// Mitsubishi GX Works2 project: 01.CumBT   PLC: FX3U/FX3UC

// global labels: Global1
VAR_GLOBAL
  Clock_Sys : INT;
  IsServer : BOOL;
  D_ReadCode : TIMER;
  D_Output : TIMER;
  OK_NG : INT;
END_VAR

FUNCTION_BLOCK Check_QR_Code
VAR_INPUT
  Req : BOOL;
END_VAR
VAR_OUTPUT
  Done : BOOL;
  Busy : BOOL;
  Error : INT;
  Trigger : BOOL;
  S_Code : INT;
END_VAR
VAR_IN_OUT
  CheckDone : BOOL;
  CfOK : INT;
END_VAR
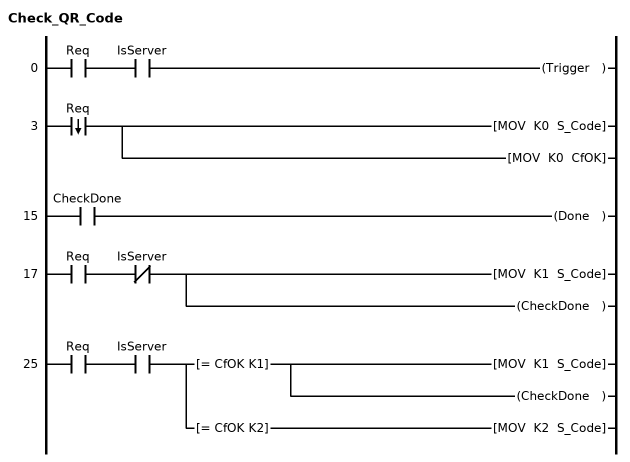
0     LD      Req
      AND     IsServer
      OUT     Trigger
3     LDF     Req
      MOV     K0 S_Code
      MOV     K0 CfOK
15    LD      CheckDone
      OUT     Done
17    LD      Req
      ANI     IsServer
      MOV     K1 S_Code
      OUT     CheckDone
25    LD      Req
      AND     IsServer
      MPS
      AND=    CfOK K1
      MOV     K1 S_Code
      OUT     CheckDone
      MPP
      AND=    CfOK K2
      MOV     K2 S_Code
END_FUNCTION_BLOCK

FUNCTION_BLOCK Control_Machine
VAR_INPUT
  AM : BOOL;
END_VAR
VAR_OUTPUT
  Red : BOOL;
  Yellow : BOOL;
  Green : BOOL;
  Buzz : BOOL;
  FlagRun : BOOL;
END_VAR
END_FUNCTION_BLOCK

FUNCTION_BLOCK Conveyer
VAR_INPUT
  AM : BOOL;
  EMG : BOOL;
END_VAR
VAR_OUTPUT
  Run_FWD : BOOL;
  Stopper_1_Up : BOOL;
  Stopper_1_Down : BOOL;
  Stopper_2_Up : BOOL;
  Stopper_2_Down : BOOL;
  Stopper_3_Up : BOOL;
  Stopper_3_Down : BOOL;
  Stopper_4_Up : BOOL;
  Stopper_4_Down : BOOL;
  XL_Up_Jig : BOOL;
  XL_Down_Jig : BOOL;
  Error_Code : INT;
END_VAR
VAR
  M_U_S1 : BOOL;
  M_D_S1 : BOOL;
  M_S_Stp1 : INT;
  M_U_S2 : BOOL;
  M_D_S2 : BOOL;
  M_S_Stp2 : INT;
  M_U_S3 : BOOL;
  M_D_S3 : BOOL;
  M_S_Stp3 : INT;
  M_U_S4 : BOOL;
  M_D_S4 : BOOL;
  M_S_Stp4 : INT;
  M_U_Jig : BOOL;
  M_D_Jig : BOOL;
  M_S_Cyl_J : INT;
  M_FWD : BOOL;
END_VAR
VAR_INPUT
  I_M_U_S1 : BOOL;
  I_M_D_S1 : BOOL;
  I_M_U_S2 : BOOL;
  I_M_D_S2 : BOOL;
  I_M_U_S3 : BOOL;
  I_M_D_S3 : BOOL;
  I_M_U_S4 : BOOL;
  I_M_D_S4 : BOOL;
  I_M_U_Jig : BOOL;
  I_M_D_Jig : BOOL;
  I_M_FWD : BOOL;
  I_M_Stop : BOOL;
END_VAR
VAR
  A_U_S1 : BOOL;
  A_D_S1 : BOOL;
  A_U_S2 : BOOL;
  A_D_S2 : BOOL;
  A_U_S3 : BOOL;
  A_D_S3 : BOOL;
  A_U_S4 : BOOL;
  A_D_S4 : BOOL;
  A_U_J : BOOL;
  A_D_J : BOOL;
END_VAR
VAR_INPUT
  A_S_Stp1 : INT;
  A_S_Stp2 : INT;
  A_S_Stp3 : INT;
  A_S_Stp4 : INT;
  A_S_Cyl_J : INT;
  A_FWD : BOOL;
END_VAR
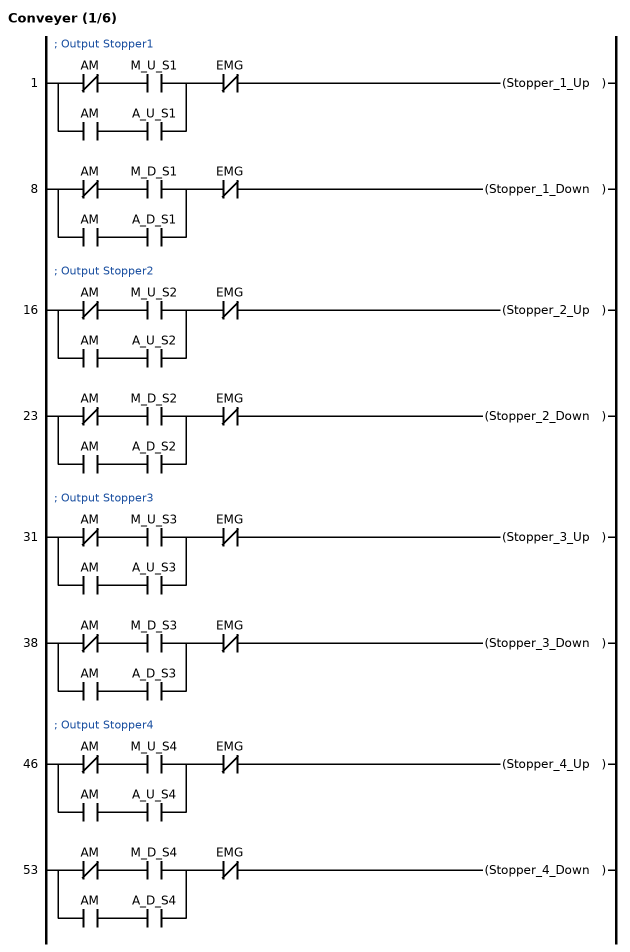
; Output Stopper1
1     LDI     AM
      AND     M_U_S1
      LD      AM
      AND     A_U_S1
      ORB
      ANI     EMG
      OUT     Stopper_1_Up
8     LDI     AM
      AND     M_D_S1
      LD      AM
      AND     A_D_S1
      ORB
      ANI     EMG
      OUT     Stopper_1_Down
; Output Stopper2
16    LDI     AM
      AND     M_U_S2
      LD      AM
      AND     A_U_S2
      ORB
      ANI     EMG
      OUT     Stopper_2_Up
23    LDI     AM
      AND     M_D_S2
      LD      AM
      AND     A_D_S2
      ORB
      ANI     EMG
      OUT     Stopper_2_Down
; Output Stopper3
31    LDI     AM
      AND     M_U_S3
      LD      AM
      AND     A_U_S3
      ORB
      ANI     EMG
      OUT     Stopper_3_Up
38    LDI     AM
      AND     M_D_S3
      LD      AM
      AND     A_D_S3
      ORB
      ANI     EMG
      OUT     Stopper_3_Down
; Output Stopper4
46    LDI     AM
      AND     M_U_S4
      LD      AM
      AND     A_U_S4
      ORB
      ANI     EMG
      OUT     Stopper_4_Up
53    LDI     AM
      AND     M_D_S4
      LD      AM
      AND     A_D_S4
      ORB
      ANI     EMG
      OUT     Stopper_4_Down
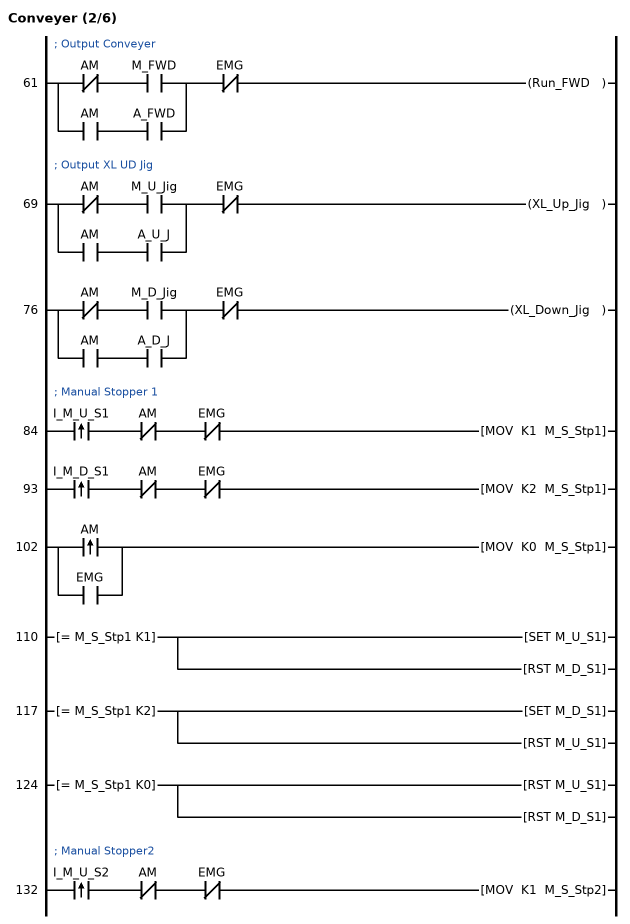
; Output Conveyer
61    LDI     AM
      AND     M_FWD
      LD      AM
      AND     A_FWD
      ORB
      ANI     EMG
      OUT     Run_FWD
; Output XL UD Jig
69    LDI     AM
      AND     M_U_Jig
      LD      AM
      AND     A_U_J
      ORB
      ANI     EMG
      OUT     XL_Up_Jig
76    LDI     AM
      AND     M_D_Jig
      LD      AM
      AND     A_D_J
      ORB
      ANI     EMG
      OUT     XL_Down_Jig
; Manual Stopper 1
84    LDP     I_M_U_S1
      ANI     AM
      ANI     EMG
      MOV     K1 M_S_Stp1
93    LDP     I_M_D_S1
      ANI     AM
      ANI     EMG
      MOV     K2 M_S_Stp1
102   LDP     AM
      OR      EMG
      MOV     K0 M_S_Stp1
110   LD=     M_S_Stp1 K1
      SET     M_U_S1
      RST     M_D_S1
117   LD=     M_S_Stp1 K2
      SET     M_D_S1
      RST     M_U_S1
124   LD=     M_S_Stp1 K0
      RST     M_U_S1
      RST     M_D_S1
; Manual Stopper2
132   LDP     I_M_U_S2
      ANI     AM
      ANI     EMG
      MOV     K1 M_S_Stp2
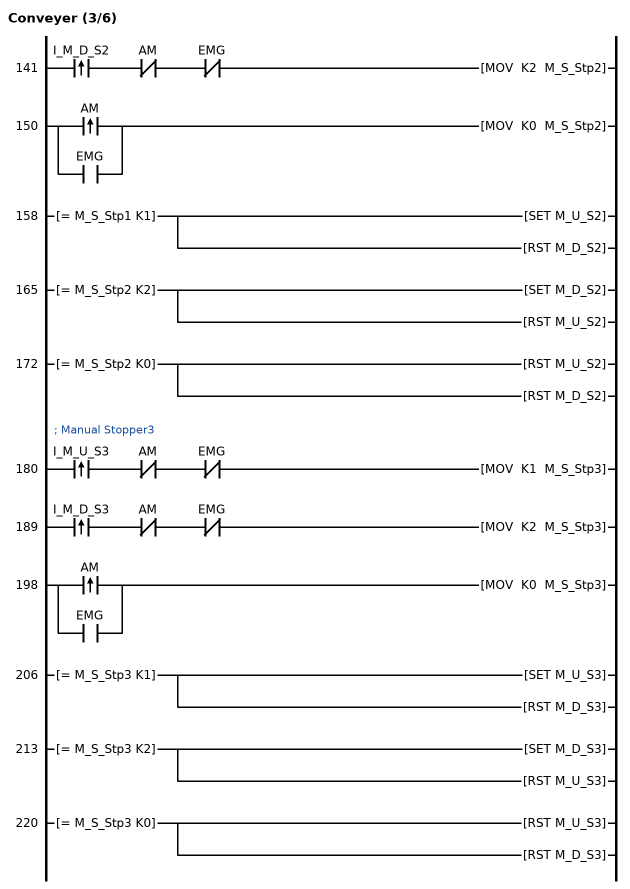
141   LDP     I_M_D_S2
      ANI     AM
      ANI     EMG
      MOV     K2 M_S_Stp2
150   LDP     AM
      OR      EMG
      MOV     K0 M_S_Stp2
158   LD=     M_S_Stp1 K1
      SET     M_U_S2
      RST     M_D_S2
165   LD=     M_S_Stp2 K2
      SET     M_D_S2
      RST     M_U_S2
172   LD=     M_S_Stp2 K0
      RST     M_U_S2
      RST     M_D_S2
; Manual Stopper3
180   LDP     I_M_U_S3
      ANI     AM
      ANI     EMG
      MOV     K1 M_S_Stp3
189   LDP     I_M_D_S3
      ANI     AM
      ANI     EMG
      MOV     K2 M_S_Stp3
198   LDP     AM
      OR      EMG
      MOV     K0 M_S_Stp3
206   LD=     M_S_Stp3 K1
      SET     M_U_S3
      RST     M_D_S3
213   LD=     M_S_Stp3 K2
      SET     M_D_S3
      RST     M_U_S3
220   LD=     M_S_Stp3 K0
      RST     M_U_S3
      RST     M_D_S3
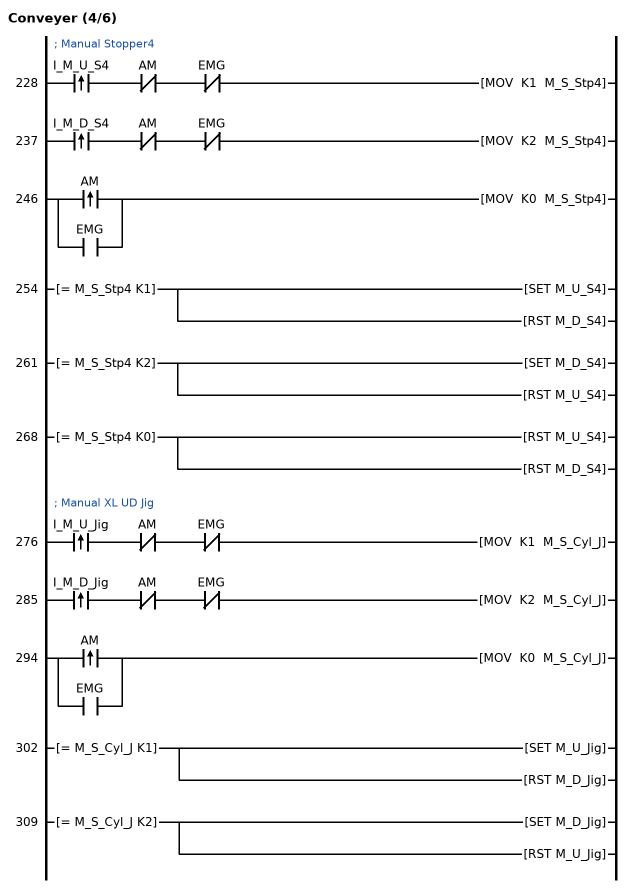
; Manual Stopper4
228   LDP     I_M_U_S4
      ANI     AM
      ANI     EMG
      MOV     K1 M_S_Stp4
237   LDP     I_M_D_S4
      ANI     AM
      ANI     EMG
      MOV     K2 M_S_Stp4
246   LDP     AM
      OR      EMG
      MOV     K0 M_S_Stp4
254   LD=     M_S_Stp4 K1
      SET     M_U_S4
      RST     M_D_S4
261   LD=     M_S_Stp4 K2
      SET     M_D_S4
      RST     M_U_S4
268   LD=     M_S_Stp4 K0
      RST     M_U_S4
      RST     M_D_S4
; Manual XL UD Jig
276   LDP     I_M_U_Jig
      ANI     AM
      ANI     EMG
      MOV     K1 M_S_Cyl_J
285   LDP     I_M_D_Jig
      ANI     AM
      ANI     EMG
      MOV     K2 M_S_Cyl_J
294   LDP     AM
      OR      EMG
      MOV     K0 M_S_Cyl_J
302   LD=     M_S_Cyl_J K1
      SET     M_U_Jig
      RST     M_D_Jig
309   LD=     M_S_Cyl_J K2
      SET     M_D_Jig
      RST     M_U_Jig
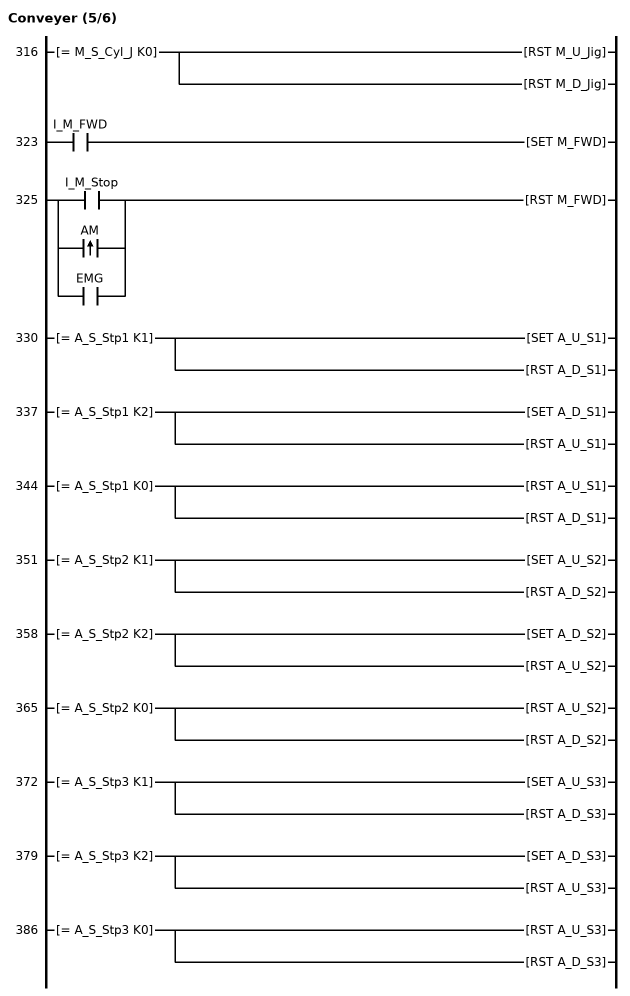
316   LD=     M_S_Cyl_J K0
      RST     M_U_Jig
      RST     M_D_Jig
323   LD      I_M_FWD
      SET     M_FWD
325   LD      I_M_Stop
      ORP     AM
      OR      EMG
      RST     M_FWD
330   LD=     A_S_Stp1 K1
      SET     A_U_S1
      RST     A_D_S1
337   LD=     A_S_Stp1 K2
      SET     A_D_S1
      RST     A_U_S1
344   LD=     A_S_Stp1 K0
      RST     A_U_S1
      RST     A_D_S1
351   LD=     A_S_Stp2 K1
      SET     A_U_S2
      RST     A_D_S2
358   LD=     A_S_Stp2 K2
      SET     A_D_S2
      RST     A_U_S2
365   LD=     A_S_Stp2 K0
      RST     A_U_S2
      RST     A_D_S2
372   LD=     A_S_Stp3 K1
      SET     A_U_S3
      RST     A_D_S3
379   LD=     A_S_Stp3 K2
      SET     A_D_S3
      RST     A_U_S3
386   LD=     A_S_Stp3 K0
      RST     A_U_S3
      RST     A_D_S3
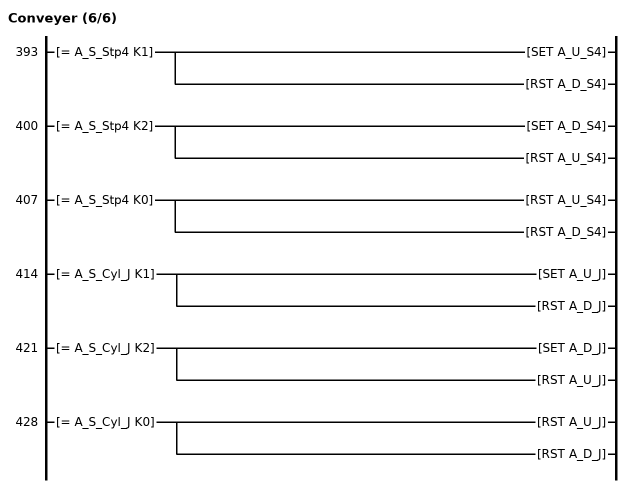
393   LD=     A_S_Stp4 K1
      SET     A_U_S4
      RST     A_D_S4
400   LD=     A_S_Stp4 K2
      SET     A_D_S4
      RST     A_U_S4
407   LD=     A_S_Stp4 K0
      RST     A_U_S4
      RST     A_D_S4
414   LD=     A_S_Cyl_J K1
      SET     A_U_J
      RST     A_D_J
421   LD=     A_S_Cyl_J K2
      SET     A_D_J
      RST     A_U_J
428   LD=     A_S_Cyl_J K0
      RST     A_U_J
      RST     A_D_J
END_FUNCTION_BLOCK

PROGRAM Data
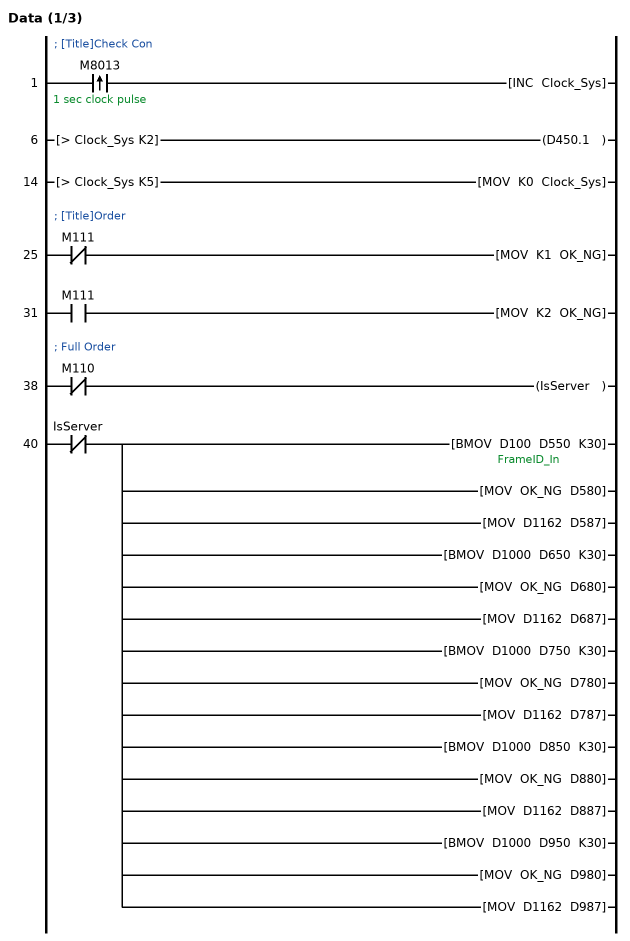
; [Title]Check Con
1     LDP     M8013  ; 1 sec clock pulse
      INC     Clock_Sys
6     LD>     Clock_Sys K2
      OUT     D450.1
14    LD>     Clock_Sys K5
      MOV     K0 Clock_Sys
; [Title]Order
25    LDI     M111
      MOV     K1 OK_NG
31    LD      M111
      MOV     K2 OK_NG
; Full Order
38    LDI     M110
      OUT     IsServer
40    LDI     IsServer
      BMOV    D100 D550 K30  ; FrameID_In
      MOV     OK_NG D580
      MOV     D1162 D587
      BMOV    D1000 D650 K30
      MOV     OK_NG D680
      MOV     D1162 D687
      BMOV    D1000 D750 K30
      MOV     OK_NG D780
      MOV     D1162 D787
      BMOV    D1000 D850 K30
      MOV     OK_NG D880
      MOV     D1162 D887
      BMOV    D1000 D950 K30
      MOV     OK_NG D980
      MOV     D1162 D987
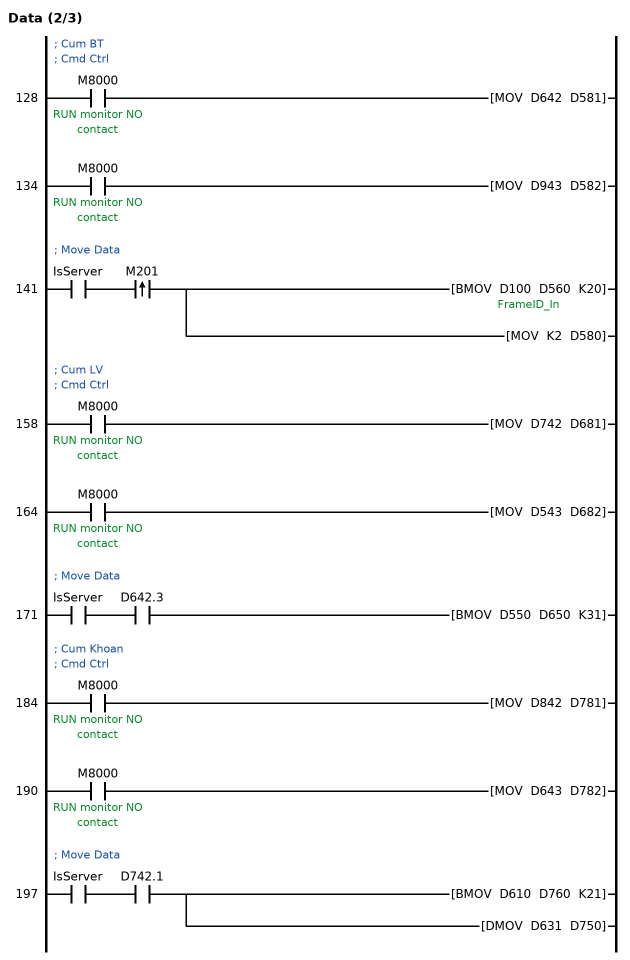
; Cum BT
; Cmd Ctrl
128   LD      M8000  ; RUN monitor NO contact
      MOV     D642 D581
134   LD      M8000  ; RUN monitor NO contact
      MOV     D943 D582
; Move Data
141   LD      IsServer
      ANDP    M201
      BMOV    D100 D560 K20
      MOV     K2 D580
; Cum LV
; Cmd Ctrl
158   LD      M8000  ; RUN monitor NO contact
      MOV     D742 D681
164   LD      M8000  ; RUN monitor NO contact
      MOV     D543 D682
; Move Data
171   LD      IsServer
      AND     D642.3
      BMOV    D550 D650 K31
; Cum Khoan
; Cmd Ctrl
184   LD      M8000  ; RUN monitor NO contact
      MOV     D842 D781
190   LD      M8000  ; RUN monitor NO contact
      MOV     D643 D782
; Move Data
197   LD      IsServer
      AND     D742.1
      BMOV    D610 D760 K21
      DMOV    D631 D750
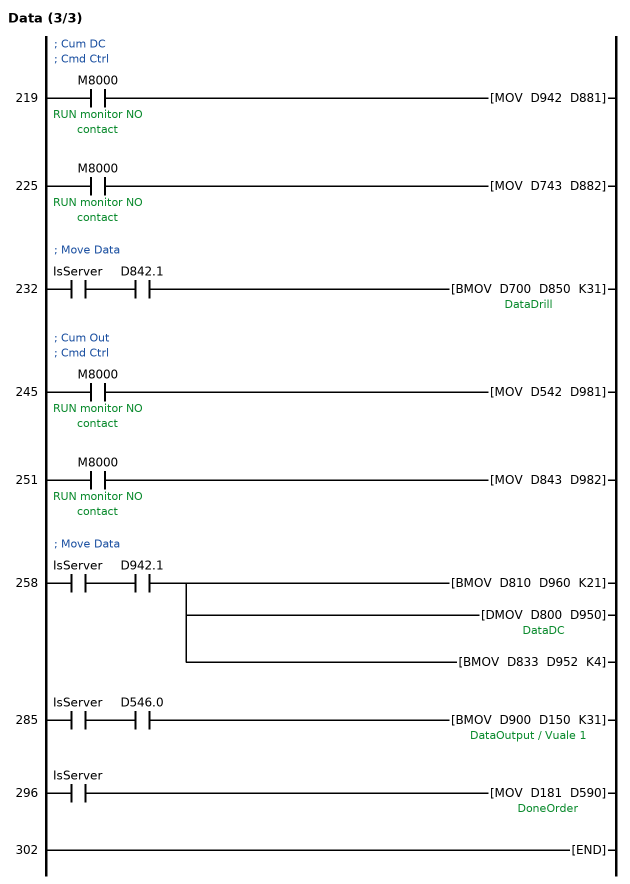
; Cum DC
; Cmd Ctrl
219   LD      M8000  ; RUN monitor NO contact
      MOV     D942 D881
225   LD      M8000  ; RUN monitor NO contact
      MOV     D743 D882
; Move Data
232   LD      IsServer
      AND     D842.1
      BMOV    D700 D850 K31  ; DataDrill
; Cum Out
; Cmd Ctrl
245   LD      M8000  ; RUN monitor NO contact
      MOV     D542 D981
251   LD      M8000  ; RUN monitor NO contact
      MOV     D843 D982
; Move Data
258   LD      IsServer
      AND     D942.1
      BMOV    D810 D960 K21
      DMOV    D800 D950  ; DataDC
      BMOV    D833 D952 K4
285   LD      IsServer
      AND     D546.0
      BMOV    D900 D150 K31  ; DataOutput / Vuale 1
296   LD      IsServer
      MOV     D181 D590  ; DoneOrder
302   END
END_PROGRAM

FUNCTION_BLOCK Fillter_Input
VAR_INPUT
  Always_True : BOOL;
END_VAR
VAR
  D_M20 : TIMER;
END_VAR
VAR_OUTPUT
  Checkout : BOOL;
END_VAR
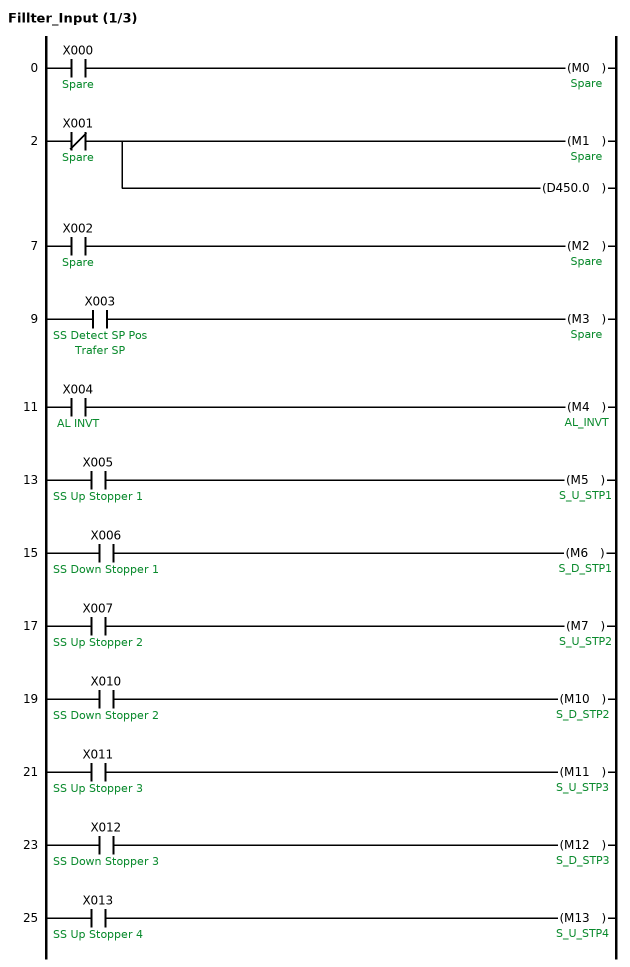
0     LD      X000  ; Spare
      OUT     M0  ; Spare
2     LDI     X001  ; Spare
      OUT     M1  ; Spare
      OUT     D450.0
7     LD      X002  ; Spare
      OUT     M2  ; Spare
9     LD      X003  ; SS Detect SP Pos Trafer SP
      OUT     M3  ; Spare
11    LD      X004  ; AL INVT
      OUT     M4  ; AL_INVT
13    LD      X005  ; SS Up Stopper 1
      OUT     M5  ; S_U_STP1
15    LD      X006  ; SS Down Stopper 1
      OUT     M6  ; S_D_STP1
17    LD      X007  ; SS Up Stopper 2
      OUT     M7  ; S_U_STP2
19    LD      X010  ; SS Down Stopper 2
      OUT     M10  ; S_D_STP2
21    LD      X011  ; SS Up Stopper 3
      OUT     M11  ; S_U_STP3
23    LD      X012  ; SS Down Stopper 3
      OUT     M12  ; S_D_STP3
25    LD      X013  ; SS Up Stopper 4
      OUT     M13  ; S_U_STP4
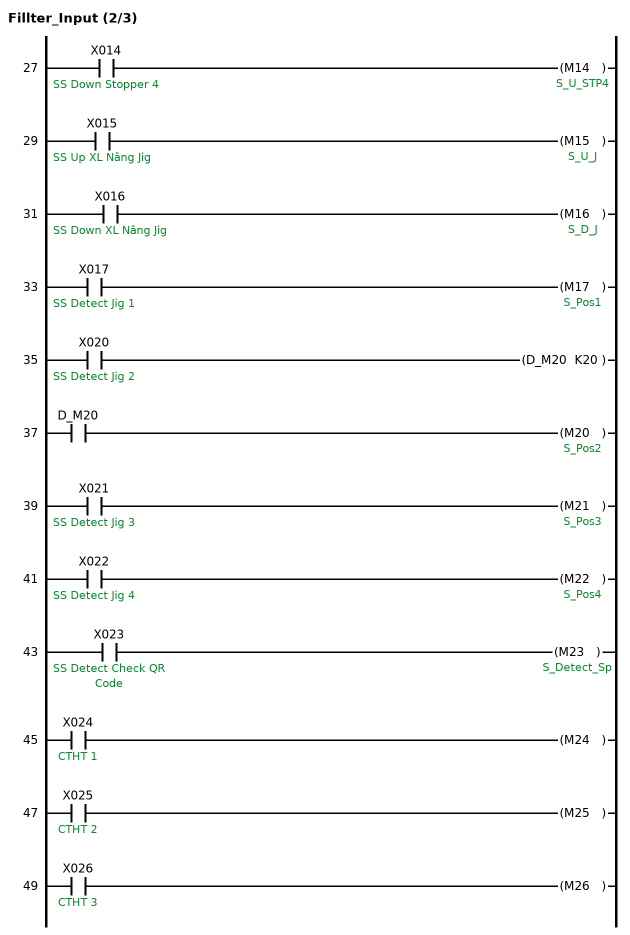
27    LD      X014  ; SS Down Stopper 4
      OUT     M14  ; S_U_STP4
29    LD      X015  ; SS Up XL Nâng Jig
      OUT     M15  ; S_U_J
31    LD      X016  ; SS Down XL Nâng Jig
      OUT     M16  ; S_D_J
33    LD      X017  ; SS Detect Jig 1
      OUT     M17  ; S_Pos1
35    LD      X020  ; SS Detect Jig 2
      OUT     D_M20 K20
37    LD      D_M20
      OUT     M20  ; S_Pos2
39    LD      X021  ; SS Detect Jig 3
      OUT     M21  ; S_Pos3
41    LD      X022  ; SS Detect Jig 4
      OUT     M22  ; S_Pos4
43    LD      X023  ; SS Detect Check QR Code
      OUT     M23  ; S_Detect_Sp
45    LD      X024  ; CTHT 1
      OUT     M24
47    LD      X025  ; CTHT 2
      OUT     M25
49    LD      X026  ; CTHT 3
      OUT     M26
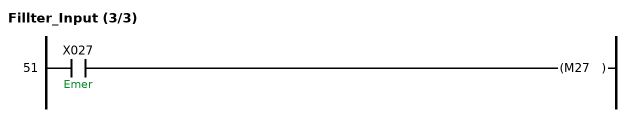
51    LD      X027  ; Emer
      OUT     M27
END_FUNCTION_BLOCK

PROGRAM MAIN
VAR
  Conveyer : Conveyer;
  Control_Machine : Control_Machine;
  Input : Fillter_Input;
  Proceduce : Proceduce;
  C_QR : Check_QR_Code;
END_VAR
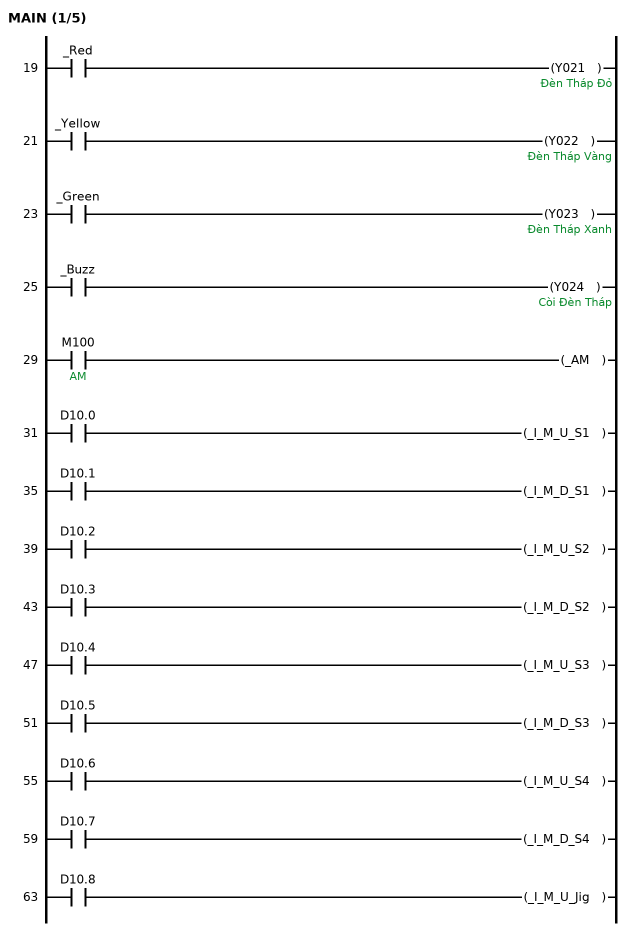
; FB BLK START Fillter_Input(Input)
; FB START
; FB_NAME Fillter_Input
; INSTANCE_NAME Input
; FB IN_B:Always_True
; FB OUT_Checkout:B
; FB END
; FB BLK END
; FB BLK START Control_Machine(Control_Machine)
; FB START
; FB_NAME Control_Machine
; INSTANCE_NAME Control_Machine
; FB IN_B:AM
; FB OUT_Red:B
; FB OUT_Yellow:B
; FB OUT_Green:B
; FB OUT_Buzz:B
; FB OUT_FlagRun:B
; FB END
19    LD      _Red
      OUT     Y021  ; Đèn Tháp Đỏ
21    LD      _Yellow
      OUT     Y022  ; Đèn Tháp Vàng
23    LD      _Green
      OUT     Y023  ; Đèn Tháp Xanh
25    LD      _Buzz
      OUT     Y024  ; Còi Đèn Tháp
; FB BLK END
; FB BLK START Conveyer(Conveyer)
29    LD      M100  ; AM
      OUT     _AM
31    LD      D10.0
      OUT     _I_M_U_S1
35    LD      D10.1
      OUT     _I_M_D_S1
39    LD      D10.2
      OUT     _I_M_U_S2
43    LD      D10.3
      OUT     _I_M_D_S2
47    LD      D10.4
      OUT     _I_M_U_S3
51    LD      D10.5
      OUT     _I_M_D_S3
55    LD      D10.6
      OUT     _I_M_U_S4
59    LD      D10.7
      OUT     _I_M_D_S4
63    LD      D10.8
      OUT     _I_M_U_Jig
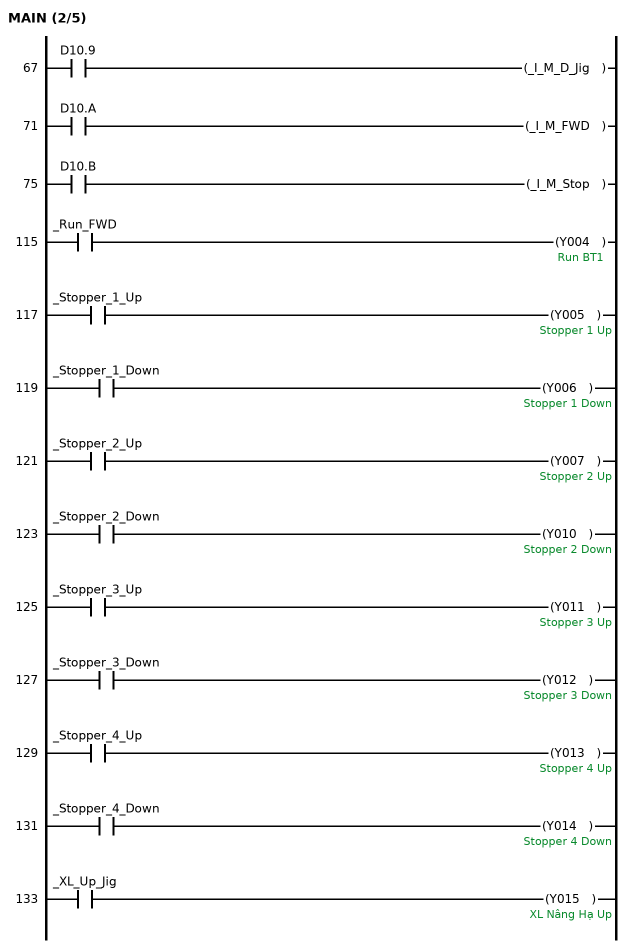
67    LD      D10.9
      OUT     _I_M_D_Jig
71    LD      D10.A
      OUT     _I_M_FWD
75    LD      D10.B
      OUT     _I_M_Stop
; FB START
; FB_NAME Conveyer
; INSTANCE_NAME Conveyer
; FB IN_B:AM
; FB OUT_Run_FWD:B
; FB IN_B:EMG
; FB OUT_Stopper_1_Up:B
; FB IN_B:I_M_U_S1
; FB OUT_Stopper_1_Down:B
; FB IN_B:I_M_D_S1
; FB OUT_Stopper_2_Up:B
; FB IN_B:I_M_U_S2
; FB OUT_Stopper_2_Down:B
; FB IN_B:I_M_D_S2
; FB OUT_Stopper_3_Up:B
; FB IN_B:I_M_U_S3
; FB OUT_Stopper_3_Down:B
; FB IN_B:I_M_D_S3
; FB OUT_Stopper_4_Up:B
; FB IN_B:I_M_U_S4
; FB OUT_Stopper_4_Down:B
; FB IN_B:I_M_D_S4
; FB OUT_XL_Up_Jig:B
; FB IN_B:I_M_U_Jig
; FB OUT_XL_Down_Jig:B
; FB IN_B:I_M_D_Jig
; FB OUT_Error_Code:W
; FB IN_B:I_M_FWD
; FB IN_B:I_M_Stop
; FB IN_W:A_S_Stp1
; FB IN_W:A_S_Stp2
; FB IN_W:A_S_Stp3
; FB IN_W:A_S_Stp4
; FB IN_W:A_S_Cyl_J
; FB IN_B:A_FWD
; FB END
115   LD      _Run_FWD
      OUT     Y004  ; Run BT1
117   LD      _Stopper_1_Up
      OUT     Y005  ; Stopper 1 Up
119   LD      _Stopper_1_Down
      OUT     Y006  ; Stopper 1 Down
121   LD      _Stopper_2_Up
      OUT     Y007  ; Stopper 2 Up
123   LD      _Stopper_2_Down
      OUT     Y010  ; Stopper 2 Down
125   LD      _Stopper_3_Up
      OUT     Y011  ; Stopper 3 Up
127   LD      _Stopper_3_Down
      OUT     Y012  ; Stopper 3 Down
129   LD      _Stopper_4_Up
      OUT     Y013  ; Stopper 4 Up
131   LD      _Stopper_4_Down
      OUT     Y014  ; Stopper 4 Down
133   LD      _XL_Up_Jig
      OUT     Y015  ; XL Nâng Hạ Up
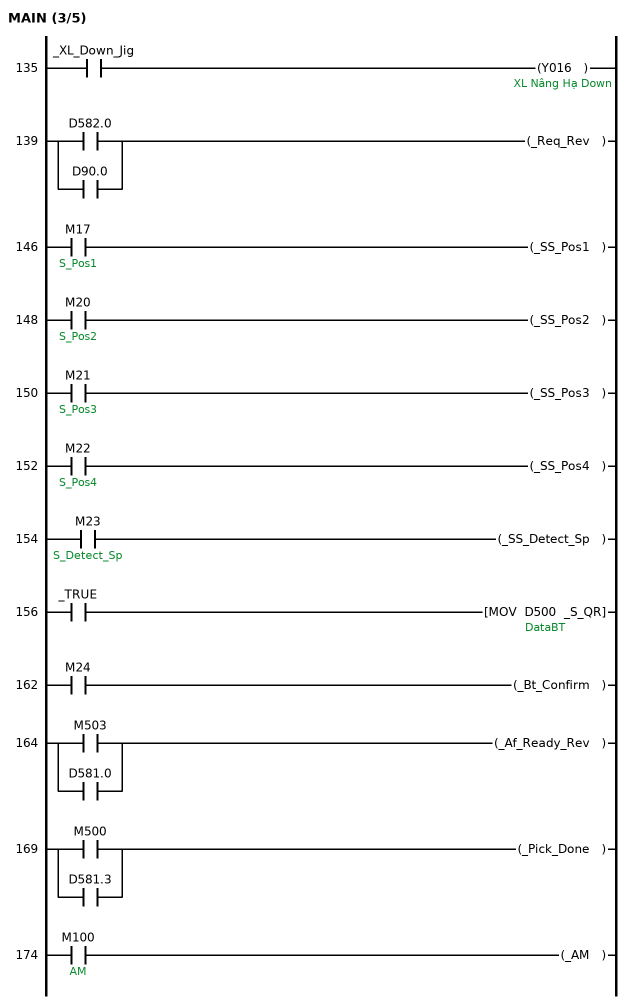
135   LD      _XL_Down_Jig
      OUT     Y016  ; XL Nâng Hạ Down
; FB BLK END
; FB BLK START Proceduce(Proceduce)
139   LD      D582.0
      OR      D90.0
      OUT     _Req_Rev
146   LD      M17  ; S_Pos1
      OUT     _SS_Pos1
148   LD      M20  ; S_Pos2
      OUT     _SS_Pos2
150   LD      M21  ; S_Pos3
      OUT     _SS_Pos3
152   LD      M22  ; S_Pos4
      OUT     _SS_Pos4
154   LD      M23  ; S_Detect_Sp
      OUT     _SS_Detect_Sp
156   LD      _TRUE
      MOV     D500 _S_QR  ; DataBT
162   LD      M24
      OUT     _Bt_Confirm
164   LD      M503
      OR      D581.0
      OUT     _Af_Ready_Rev
169   LD      M500
      OR      D581.3
      OUT     _Pick_Done
174   LD      M100  ; AM
      OUT     _AM
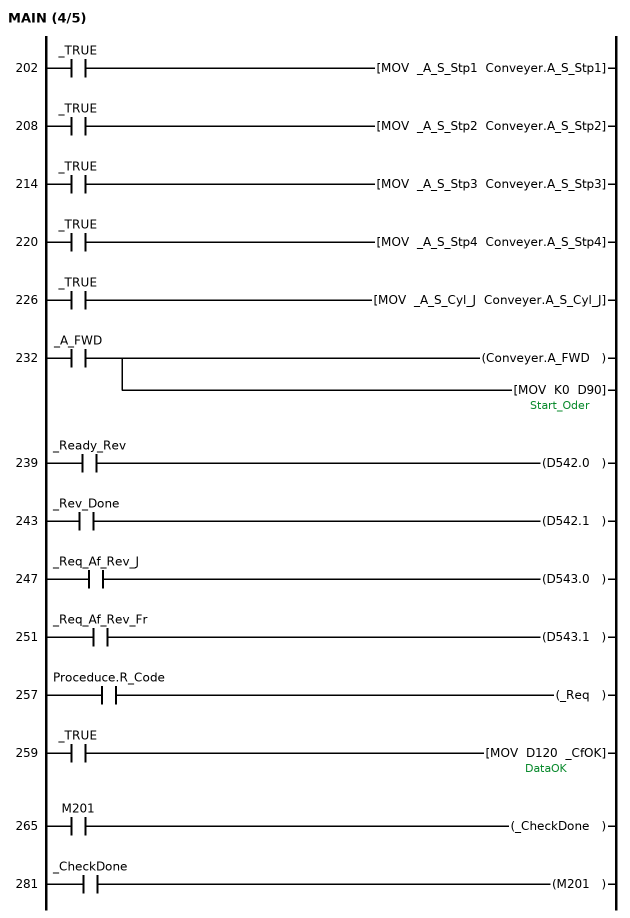
; FB START
; FB_NAME Proceduce
; INSTANCE_NAME Proceduce
; FB IN_B:Req_Rev
; FB OUT_A_S_Stp1:W
; FB IN_B:SS_Pos1
; FB OUT_A_S_Stp2:W
; FB IN_B:SS_Pos2
; FB OUT_A_S_Stp3:W
; FB IN_B:SS_Pos3
; FB OUT_A_S_Stp4:W
; FB IN_B:SS_Pos4
; FB OUT_A_S_Cyl_J:W
; FB IN_B:SS_Detect_Sp
; FB OUT_A_FWD:B
; FB IN_W:S_QR
; FB OUT_R_Code:B
; FB IN_B:Bt_Confirm
; FB OUT_Ready_Rev:B
; FB IN_B:Af_Ready_Rev
; FB OUT_Rev_Done:B
; FB IN_B:Pick_Done
; FB OUT_Req_Af_Rev_J:B
; FB IN_B:AM
; FB OUT_Req_Af_Rev_Fr:B
; FB END
202   LD      _TRUE
      MOV     _A_S_Stp1 Conveyer.A_S_Stp1
208   LD      _TRUE
      MOV     _A_S_Stp2 Conveyer.A_S_Stp2
214   LD      _TRUE
      MOV     _A_S_Stp3 Conveyer.A_S_Stp3
220   LD      _TRUE
      MOV     _A_S_Stp4 Conveyer.A_S_Stp4
226   LD      _TRUE
      MOV     _A_S_Cyl_J Conveyer.A_S_Cyl_J
232   LD      _A_FWD
      OUT     Conveyer.A_FWD
      MOV     K0 D90  ; Start_Oder
239   LD      _Ready_Rev
      OUT     D542.0
243   LD      _Rev_Done
      OUT     D542.1
247   LD      _Req_Af_Rev_J
      OUT     D543.0
251   LD      _Req_Af_Rev_Fr
      OUT     D543.1
; FB BLK END
; FB BLK START Check_QR_Code(C_QR)
257   LD      Proceduce.R_Code
      OUT     _Req
259   LD      _TRUE
      MOV     D120 _CfOK  ; DataOK
265   LD      M201
      OUT     _CheckDone
; FB START
; FB_NAME Check_QR_Code
; INSTANCE_NAME C_QR
; FB IN_B:Req
; FB OUT_CfOK:W
; FB IN_W:CfOK
; FB OUT_CheckDone:B
; FB IN_B:CheckDone
; FB OUT_Trigger:B
; FB OUT_Done:B
; FB OUT_Busy:B
; FB OUT_Error:W
; FB OUT_S_Code:W
; FB END
281   LD      _CheckDone
      OUT     M201
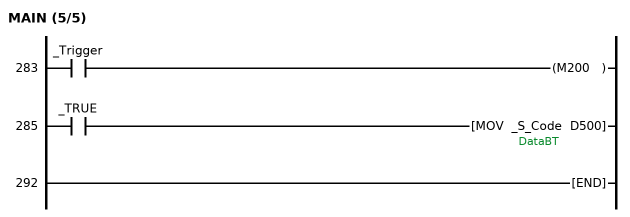
283   LD      _Trigger
      OUT     M200
285   LD      _TRUE
      MOV     _S_Code D500
; FB BLK END
292   END
END_PROGRAM

FUNCTION_BLOCK Proceduce
VAR_INPUT
  Req_Rev : BOOL;
END_VAR
VAR_OUTPUT
  A_S_Stp1 : INT;
  A_S_Stp2 : INT;
  A_S_Stp3 : INT;
  A_S_Stp4 : INT;
  A_S_Cyl_J : INT;
  A_FWD : BOOL;
END_VAR
VAR_INPUT
  SS_Pos1 : BOOL;
  SS_Pos2 : BOOL;
  SS_Pos3 : BOOL;
  SS_Pos4 : BOOL;
  SS_Detect_Sp : BOOL;
END_VAR
VAR_OUTPUT
  R_Code : BOOL;
END_VAR
VAR_INPUT
  S_QR : INT;  (* 1: OK 2:NG 0:No S *)
END_VAR
VAR
  A_R_TH1 : BOOL;
  A_R_TH2 : BOOL;
END_VAR
VAR_INPUT
  Bt_Confirm : BOOL;
END_VAR
VAR
  A_R_TH3 : BOOL;
  A_R_TH4 : BOOL;
  A_R_TH5 : BOOL;
END_VAR
VAR_INPUT
  Af_Ready_Rev : BOOL;
  Pick_Done : BOOL;
END_VAR
VAR
  Limit_R : TIMER;
END_VAR
VAR_INPUT
  AM : BOOL;
END_VAR
VAR_OUTPUT
  Ready_Rev : BOOL;
  Rev_Done : BOOL;
  Req_Af_Rev_J : BOOL;
  Req_Af_Rev_Fr : BOOL;
END_VAR
VAR
  D_Req_Rev_Fr : TIMER;
END_VAR
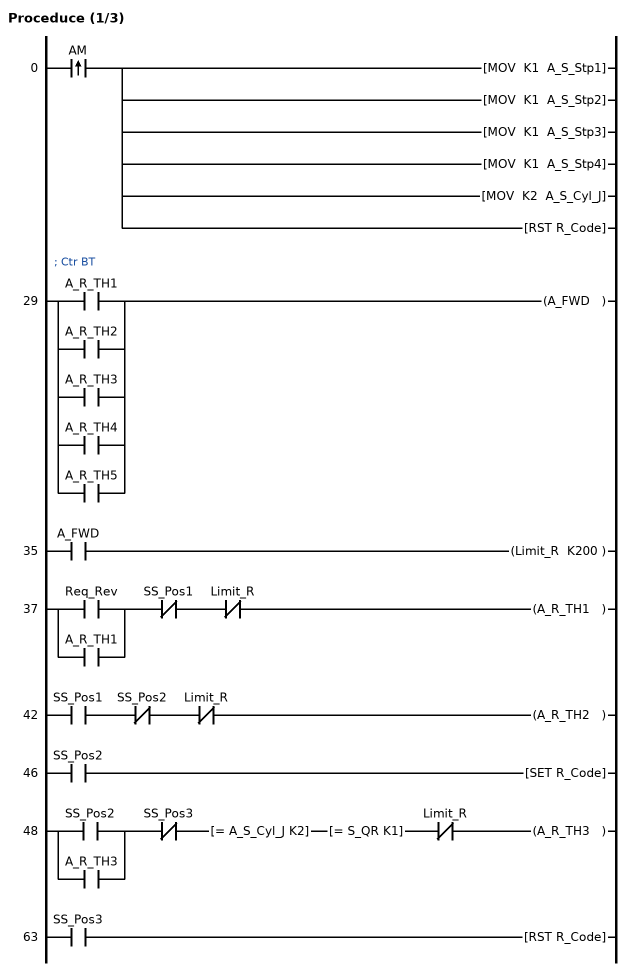
0     LDP     AM
      MOV     K1 A_S_Stp1
      MOV     K1 A_S_Stp2
      MOV     K1 A_S_Stp3
      MOV     K1 A_S_Stp4
      MOV     K2 A_S_Cyl_J
      RST     R_Code
; Ctr BT
29    LD      A_R_TH1
      OR      A_R_TH2
      OR      A_R_TH3
      OR      A_R_TH4
      OR      A_R_TH5
      OUT     A_FWD
35    LD      A_FWD
      OUT     Limit_R K200
37    LD      Req_Rev
      OR      A_R_TH1
      ANI     SS_Pos1
      ANI     Limit_R
      OUT     A_R_TH1
42    LD      SS_Pos1
      ANI     SS_Pos2
      ANI     Limit_R
      OUT     A_R_TH2
46    LD      SS_Pos2
      SET     R_Code
48    LD      SS_Pos2
      OR      A_R_TH3
      ANI     SS_Pos3
      AND=    A_S_Cyl_J K2
      AND=    S_QR K1
      ANI     Limit_R
      OUT     A_R_TH3
63    LD      SS_Pos3
      RST     R_Code
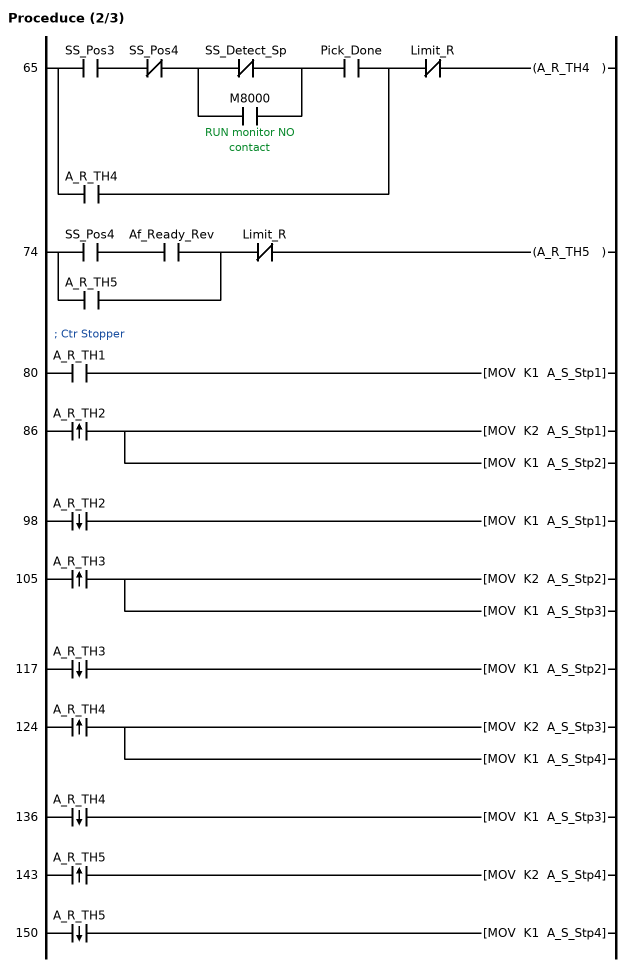
65    LD      SS_Pos3
      ANI     SS_Pos4
      LDI     SS_Detect_Sp
      OR      M8000  ; RUN monitor NO contact
      ANB
      AND     Pick_Done
      OR      A_R_TH4
      ANI     Limit_R
      OUT     A_R_TH4
74    LD      SS_Pos4
      AND     Af_Ready_Rev
      OR      A_R_TH5
      ANI     Limit_R
      OUT     A_R_TH5
; Ctr Stopper
80    LD      A_R_TH1
      MOV     K1 A_S_Stp1
86    LDP     A_R_TH2
      MOV     K2 A_S_Stp1
      MOV     K1 A_S_Stp2
98    LDF     A_R_TH2
      MOV     K1 A_S_Stp1
105   LDP     A_R_TH3
      MOV     K2 A_S_Stp2
      MOV     K1 A_S_Stp3
117   LDF     A_R_TH3
      MOV     K1 A_S_Stp2
124   LDP     A_R_TH4
      MOV     K2 A_S_Stp3
      MOV     K1 A_S_Stp4
136   LDF     A_R_TH4
      MOV     K1 A_S_Stp3
143   LDP     A_R_TH5
      MOV     K2 A_S_Stp4
150   LDF     A_R_TH5
      MOV     K1 A_S_Stp4
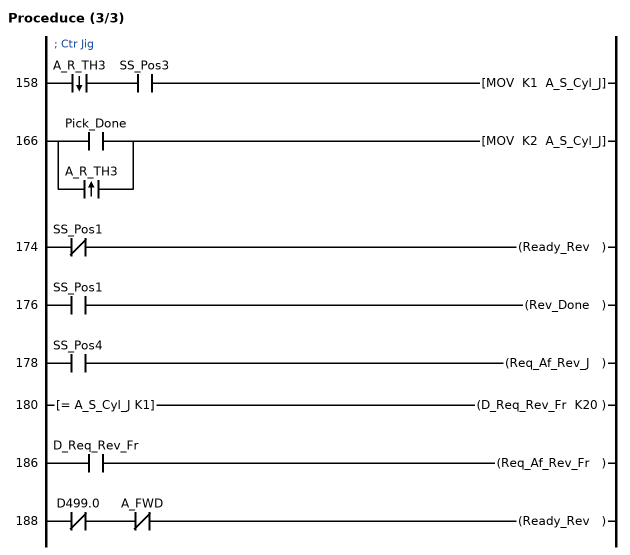
; Ctr Jig
158   LDF     A_R_TH3
      AND     SS_Pos3
      MOV     K1 A_S_Cyl_J
166   LD      Pick_Done
      ORP     A_R_TH3
      MOV     K2 A_S_Cyl_J
174   LDI     SS_Pos1
      OUT     Ready_Rev
176   LD      SS_Pos1
      OUT     Rev_Done
178   LD      SS_Pos4
      OUT     Req_Af_Rev_J
180   LD=     A_S_Cyl_J K1
      OUT     D_Req_Rev_Fr K20
186   LD      D_Req_Rev_Fr
      OUT     Req_Af_Rev_Fr
188   LDI     D499.0
      ANI     A_FWD
      OUT     Ready_Rev
END_FUNCTION_BLOCK

PROGRAM ALARM
0     END
END_PROGRAM

// device comments not shown above
M220  ; TriggerrQr
D152  ; Value 2
D154  ; Vuale 3
D156  ; Value 4
D158  ; Value 5
D160  ; FrameID_Out
D180  ; StatusFrame
D600  ; DataLV
